(* Schneider Machine Expert - Basic project Bloc Fonction Compteur et PWM, file version 1.2.0.0 *)

HARDWARE
  Cpu 0: TM221ME16T/G
  EthernetConfiguration: NetworkName=M221, IpAllocationMode=FixedAddress, IpAddress=10.10.1.135, SubnetMask=255.255.255.0
  SerialLineConfiguration: Baud=Baud19200, Parity=ParityEven, DataBits=DataBits8, StopBits=StopBits1, PhysicalMedium=PhysicalMediumRs485, TransmissionMode=TransmissionModeModbusRtu, SlaveId=1, Addressing=SlaveAddressing
  MastTask: UsePeriodScanMode=false, PeriodScan=100
  FastTask: Period=255
  CpuBehavior: StartingMode=StartInRun, AutoSaveRamOnEeprom=true, WatchdogPeriod=250

SYMBOLS  (address, symbol, comment, settings)
  %M1       TROISSEC
  %M2       SENS_COMPTAGE
  %HSC0       [Type=SimpleCounter, Preset=0, ThresholdS0=3000, DedicatedInputs(DedicatedInput(Activated=true, IsAvailable=true), DedicatedInput(IsAvailable=true), DedicatedInput(Editable=true, IsAvailable=true), DedicatedInput(Editable=true, IsAvailable=true)), ReflexOutputs(ReflexOutput(Activated=false, LessThanS0=false, GreaterOrEqualThanS0=false, GreaterOrEqualThanS1=false, Editable=true), ReflexOutput(Activa]
  %PWM0     GÉNÉRATEUR_DIMPULSION  [GlobalIndex=0, Type=PWM, TimeBase=OneMilliSeconds, Preset=1]

POU Nouveau POU
  (* SectionNumber=1, IsGrafcet=false *)

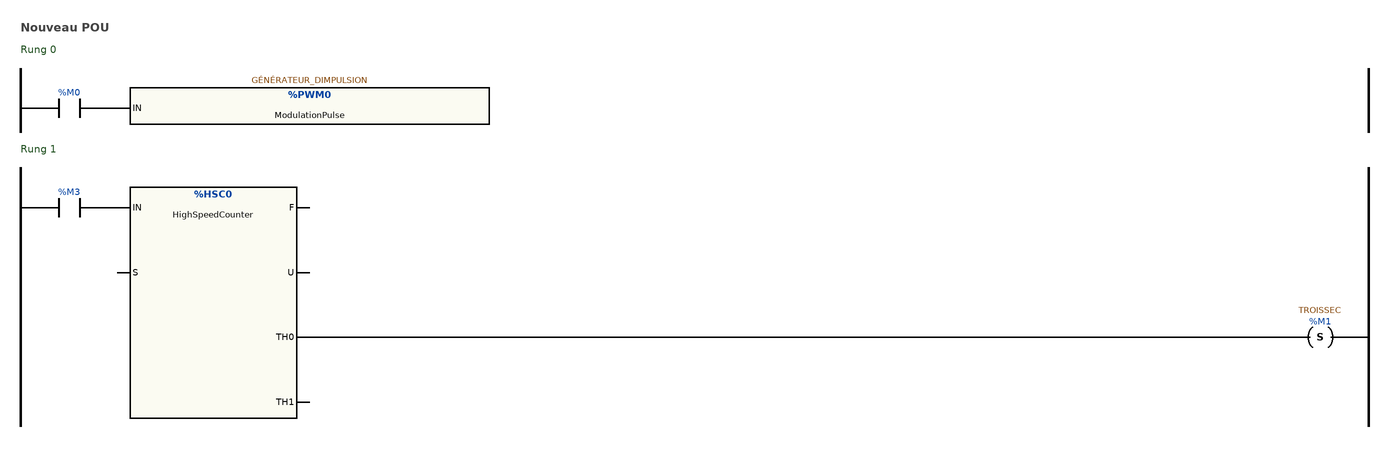

// Rung 0
  BLK %PWM0               (* GÉNÉRATEUR_DIMPULSION *)
  LD %M0
  IN
  END_BLK
  // as ST:
  //   GÉNÉRATEUR_DIMPULSION(IN := %M0);

// Rung 1
  BLK %HSC0
  LD %M3
  IN
  OUT_BLK
  LD TH0
  S %M1                   (* TROISSEC *)
  END_BLK
  // as ST:
  //   %HSC0(IN := %M3);
  //   IF %HSC0.TH0 THEN TROISSEC := TRUE; END_IF;
